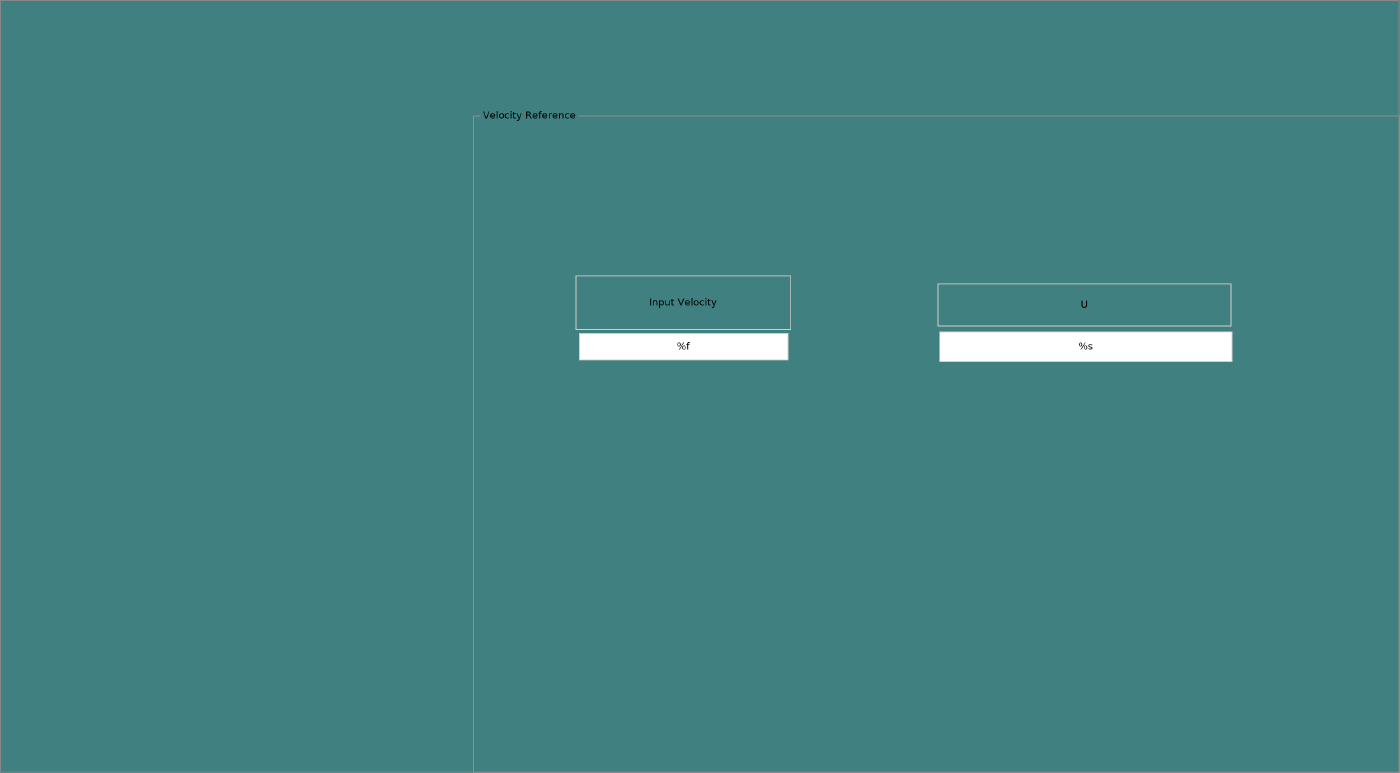
VISUALIZATION OpenLoopTest  // 1574x870
    GroupBox (532,122 1042x748), "Velocity Reference"
        Textfield (119,253 235x30), "%f", text variable: G_Parameters.stParam.V_ref
            OnMouseClick: write the text variable via Default
        Textfield (524,251 329x34), "%s", text variable: G_Parameters.stParam.U
        Textfield (115,188 242x61), "Input Velocity"
        Textfield (522,197 330x48), "U"
END_VISUALIZATION

(* stored: Version 1.1.0.1, ProductVersion 3.1.4024.12
   Visu OpenLoopTest: Id {da5bfb05-2e82-4333-86a6-45b0f170f4fe} *)
